{attribute 'linkalways'} 
{attribute 'no_explicit_call' := 'This FB is a CLASS and must be accessed using methods or properties'}
{attribute 'enable_dynamic_creation'}
FUNCTION_BLOCK Node_F_VN_ImageAverageStdDev EXTENDS VisionNode
VAR
    ipSrcImage : _ITcVnImage;
    aAverage : _TcVnVector4_LREAL;
    aStdDev : _TcVnVector4_LREAL;
    hrPrev : _HRESULT(S_OK);
	hresult : _HRESULT(S_OK);
END_VAR

METHOD PUBLIC  Clone : I_Node
VAR
	pNode : POINTER TO Node_F_VN_ImageAverageStdDev;
END_VAR
pNode := __NEW(Node_F_VN_ImageAverageStdDev);
Clone := pNode^;
END_METHOD

METHOD FB_init : BOOL
VAR_INPUT
	bInitRetains : BOOL; // if TRUE, the retain variables are initialized (warm start / cold start)
	bInCopyCode : BOOL;  // if TRUE, the instance afterwards gets moved into the copy code (online change)
END_VAR
AddInput('ipSrcImage', ipSrcImage);
AddInput('hrPrev', hrPrev);
AddOutput('aAverage', aAverage);
AddOutput('aStdDev', aStdDev);
AddOutput('hresult', hresult);
END_METHOD

METHOD PROTECTED OnExecute
hresult.Value := F_VN_ImageAverageStdDev(
	ipSrcImage := ipSrcImage.Value,
    aAverage := aAverage.Value,
    aStdDev := aStdDev.Value,
	hrPrev:= hrPrev.Value);
END_METHOD

METHOD PUBLIC PreExecutionCheck
VAR_INPUT
	Check : I_PreExecutionChecks;
END_VAR
Check.IsTrue(ipSrcImage.IsValid, 'ipSrcImage must contain an image');
Check.IsTrue((ipSrcImage.HasChannelCount(1) OR
              ipSrcImage.HasChannelCount(2) OR
              ipSrcImage.HasChannelCount(3) OR
              ipSrcImage.HasChannelCount(4)), 'ipSrcImage must contain 1, 2, 3 or 4 channels');
END_METHOD

END_FUNCTION_BLOCK

(* stored: Version 1.1.0.1, ProductVersion 3.1.4024.13
   POU Node_F_VN_ImageAverageStdDev: Id {62a6c6d6-1ac6-0925-3b9f-36ce6c5ef541}, SpecialFunc None
   Folder Constructor: Id {e67369d6-d935-0a93-2095-821f7d7dd5fa}
   Method Clone: Id {d087c1fd-a34c-0a47-3858-cfd5a23cbb4a}
   Method FB_init: Id {b67aa782-c5f3-0b96-110d-f34ea605d15d}
   Method OnExecute: Id {bb429bc7-8d81-0236-1fba-79367fc81a4f}
   Method PreExecutionCheck: Id {cd83f059-01dc-0b1d-0c9f-6aef6bad6f17} *)
